PROGRAM MAIN
VAR
END_VAR

END_PROGRAM

(* stored: Version 1.1.0.1
   POU MAIN: Id {9b29ec95-2a4a-4ce6-b11d-44b036dedb9e} *)
